// TIA Portal V20 export
DATA_BLOCK "Data"   // DB40
{ S7_Optimized_Access := 'TRUE' }
// stored: MemoryReserve 100
   VAR
      general : "LAF_typeGeneralStatus";
   END_VAR
BEGIN
   general.simulation.plcInternal := TRUE;
   // general.enablePower : Global power is off
END_DATA_BLOCK
